{attribute 'qualified_only'}
{attribute 'strict'}
{attribute 'to_string'}
TYPE EMppcStateModule :
(
	UNRECOVERABLE_ERROR := 0,
	AWAITING_COOLING_TEMP_STABLE,
	AWAITING_HIGH_VOLTAGE_POWER_SUPPLY_STABLE,
	MODULE_OPERATING_NORMAL 
);
END_TYPE

(* stored: Version 1.1.0.1, ProductVersion 3.1.4024.4
   DUT EMppcStateModule: Id {bfcfe603-bf32-466f-b5b9-8e1d8228cfa3} *)
